FUNCTION_BLOCK FlowInput EXTENDS AnalogInput
VAR_INPUT
	k: LREAL;
END_VAR
VAR_OUTPUT
END_VAR
VAR
	Aver: Average;
END_VAR
VAR PERSISTENT
END_VAR

SUPER^();

METHOD FB_init : BOOL
VAR_INPUT
	bInitRetains : BOOL; // if TRUE, the retain variables are initialized (warm start / cold start)
	bInCopyCode : BOOL;  // if TRUE, the instance afterwards gets moved into the copy code (online change)
END_VAR
IF bInitRetains THEN
	ProcessMin := 0;
	ProcessMax := 30000;
	MinValue := 0;
	MaxValue := 30000;
END_IF
END_METHOD

METHOD GetValue : LREAL
VAR_INPUT
END_VAR
VAR
	Pressure: LREAL;
END_VAR
Pressure := SUPER^.GetValue();
Aver(NewSample := PressureToFlow(Pressure, k));
GetValue := Aver.Value;
END_METHOD

END_FUNCTION_BLOCK

(* stored: Version 1.1.0.1, ProductVersion 3.1.4024.6
   POU FlowInput: Id {252a420b-3d35-42f1-8b50-a89741fad6f9}, SpecialFunc None
   Method FB_init: Id {b79f8368-e24f-4edd-a475-486dea9c9596}
   Method GetValue: Id {c48d5cf9-d7a8-4783-8146-858a11b9064d} *)
